TYPE ST_AxisParameter :
STRUCT
	Velocity : LREAL;
	Acceleration : LREAL;
	Deceleration : LREAL;
	Jerk : LREAL;
END_STRUCT
END_TYPE

(* stored: Version 1.1.0.1, ProductVersion 3.1.4026.6
   DUT ST_AxisParameter: Id {73c28d29-da91-477d-9329-73849d5d9d27} *)
